Omron CX-Programmer project NewProject (CX-Programmer 9.75)

# PLC OMRON: CP1E N30

## Global symbols (name address type ; comment)
C001 BOOL  ; C1
T001 BOOL  ; T1
T002 BOOL  ; T2
T003 BOOL  ; T3
T004 BOOL  ; T4
T005 BOOL  ; T5
T006 BOOL  ; T6

## Program NewProgram1 (cyclic task 0)
Local symbols
ConveyMotor 100.05 BOOL  ; 100.05
MainSupply 100.00 BOOL  ; 100.00
MixingMotor 100.03 BOOL  ; 100.03
Restart 100.06 BOOL  ; 100.06
Start 0.00 BOOL  ; 0.00
Stop 0.01 BOOL  ; 0.01
V1 100.01 BOOL  ; 100.01
V2 100.02 BOOL  ; 100.02
V3 100.04 BOOL  ; 100.04

### Section Section1

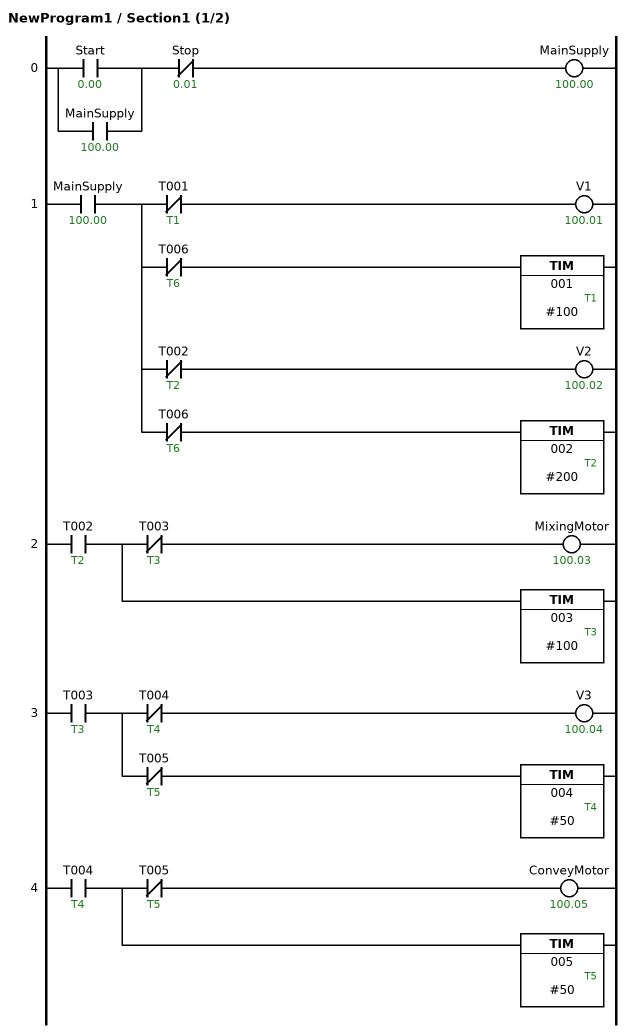
; rung 0
LD Start  ; 0.00
OR MainSupply  ; 100.00
ANDNOT Stop  ; 0.01
OUT MainSupply  ; 100.00
; rung 1
LD MainSupply  ; 100.00
OUT TR0
ANDNOT T001  ; T1
OUT V1  ; 100.01
LD TR0
ANDNOT T006  ; T6
TIM 001 #100  ; T1
LD TR0
ANDNOT T002  ; T2
OUT V2  ; 100.02
LD TR0
ANDNOT T006  ; T6
TIM 002 #200  ; T2
; rung 2
LD T002  ; T2
OUT TR0
ANDNOT T003  ; T3
OUT MixingMotor  ; 100.03
LD TR0
TIM 003 #100  ; T3
; rung 3
LD T003  ; T3
OUT TR0
ANDNOT T004  ; T4
OUT V3  ; 100.04
LD TR0
ANDNOT T005  ; T5
TIM 004 #50  ; T4
; rung 4
LD T004  ; T4
OUT TR0
ANDNOT T005  ; T5
OUT ConveyMotor  ; 100.05
LD TR0
TIM 005 #50  ; T5

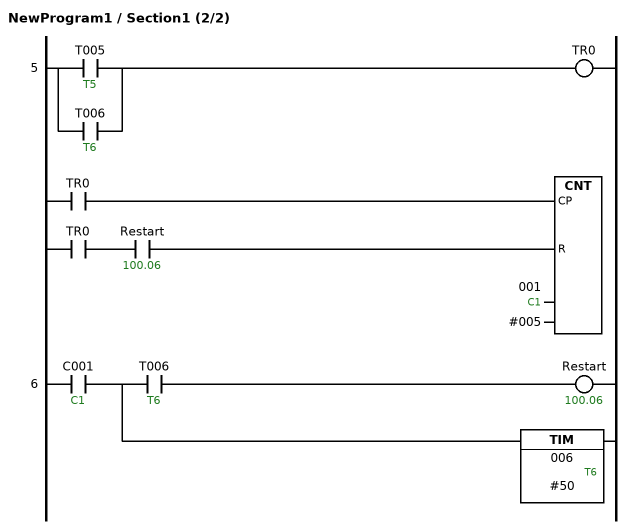
; rung 5
LD T005  ; T5
OR T006  ; T6
OUT TR0
LD TR0
AND Restart  ; 100.06
CNT 001 #005  ; C1
; rung 6
LD C001  ; C1
OUT TR0
AND T006  ; T6
OUT Restart  ; 100.06
LD TR0
TIM 006 #50  ; T6

### Section END
; rung 0
END(001)